{attribute 'qualified_only'}
{attribute 'strict'}
{attribute 'to_string'}
TYPE
    eMachineModes :
    (
        Idle    := 0,
        Automat := 1000,
        Step    := 2000,
        Home    := 3000,
        Manual  := 4000,
        Fault   := 9000
    ) INT;
END_TYPE

(* stored: Version 1.1.0.1, ProductVersion 3.1.4024.12
   DUT eMachineModes: Id {b4fbe22c-264d-0c3f-041a-83b8aad68a05} *)
